(* PLC project Aufgabe2SPS, Beckhoff Automation GmbH TwinCAT PLC Control 3.5.13.20 *)
(* stored: creationDateTime 2020-03-31T15:44:23.6339566, modificationDateTime 2020-03-31T15:44:23.6389422 *)

TYPE ST_STATUS_WORD_DATA :
STRUCT
	inLenght : INT;
   overrunError  :  BOOL;
   framingError  :  BOOL;
   parityError  :  BOOL;
   bufferFull  :  BOOL;
   initAccepted  :  BOOL;
   receiveRequest  :  BOOL;
   transmitAccepted  :  BOOL;		

END_STRUCT
END_TYPE

TYPE ST_CurrentStatus :
STRUCT
	buttonYellow : BOOL;
	buttonBlue : BOOL;
	// usw...
END_STRUCT
END_TYPE

FUNCTION_BLOCK FB_EdgeDetector
VAR_INPUT
	b_InputSignal_k : BOOL;
END_VAR
VAR_OUTPUT
	b_PositiveEdge : BOOL;
	b_NegativeEdge : BOOL;
END_VAR
VAR
	b_InputSignal_k_1 : BOOL;
END_VAR

                  b_PositiveEdge := b_InputSignal_k AND NOT b_InputSignal_k_1;
b_NegativeEdge := NOT b_InputSignal_k AND b_InputSignal_k_1;

b_InputSignal_k_1 := b_InputSignal_k;
                
END_FUNCTION_BLOCK

FUNCTION F_AdditionFunction : INT
VAR_INPUT
	i_var1 : INT;
	i_var2 : INT;
END_VAR
VAR
	
END_VAR

                  F_AdditionFunction := i_var1 + i_var2;
                
END_FUNCTION

FUNCTION F_DivisionFunction : INT
VAR_INPUT
	i_var1 : INT;
	i_var2 : INT;
END_VAR
VAR
	
END_VAR

                  IF i_var2 = 0 THEN
	F_DivisionFunction := 0;
ELSE	
	F_DivisionFunction := i_var1 / i_var2;
END_IF

                
END_FUNCTION

FUNCTION F_STATUS_WORD_PROC : ST_STATUS_WORD_DATA
VAR_INPUT
	w_StatusWord : WORD;
END_VAR
VAR
END_VAR

                  

F_STATUS_WORD_PROC.transmitAccepted := w_StatusWord.0;
F_STATUS_WORD_PROC.parityError := w_StatusWord.1;
F_STATUS_WORD_PROC.initAccepted := w_StatusWord.2;
F_STATUS_WORD_PROC.bufferFull := w_StatusWord.3;
F_STATUS_WORD_PROC.parityError := w_StatusWord.4;
F_STATUS_WORD_PROC.framingError := w_StatusWord.5;
F_STATUS_WORD_PROC.overrunError := w_StatusWord.6;
F_STATUS_WORD_PROC.inLenght := WORD_TO_INT(SHR(w_StatusWord,8));
                
END_FUNCTION

PROGRAM MAIN
VAR
	// Lokale Variablen um die Funktionen
	// F_AdditionFunction und F_DivisionFunction zu testen
	i_var1   : INT;
	i_var2   : INT;
	i_addRes : INT;
	i_divRes : INT;
	
	// 16 bits
	w_myword : WORD := 16#5D7A;
	w_divRes : WORD;
	
	// 32 bits
	dw_mydword : DWORD;
	dw_mydword1 : DWORD;
	
	w_testWord : WORD;
	
	st_resRsProt : ST_STATUS_WORD_DATA;
	
	// Array von REAL, Dimension 10
	// arr_r_testArray : ARRAY[0..9] OF REAL;
	arr_r_testArray : ARRAY[1..10] OF REAL;
	
	// Variablen für FOR Schleife
	r_SummeArray : REAL;
	r_MulArray : REAL;
	
	// Variabel für FOR Schleife
	i_SchleifeIterVar : INT;
	
	// Edge detektor 2 Mal instanzieren
	fbEdgeDetectorGelb : FB_EdgeDetector;
	fbEdgeDetectorBlau : FB_EdgeDetector;
	
	// "Software" Taster um Edge Detektor zu testen
	bGelbTaster : BOOL;
	bBlauTaster : BOOL;
	
	// "Software" Leucthmelder
	bRedLight : BOOL;
	bGreenLight : BOOL;
	
	// Steuerbefehle für die Lampen
	bCommandForLights : BOOL := FALSE;
	
	// Number of Zyklen in 1/3 Sekunde (3 Hz)
	uiTicksNumber3Herz : UINT := 0;
	
	// Zähler
	uiTicksCounter : UINT := 0;
	
	// TRUE if positive Flanke bei gelbem Taster
	bGelbPositivEdge : BOOL;
	
	// Mittelwert vom Signal ***************
	rMeanVoltageValue : REAL;
	// Über die letzten 100 Werten
	rMeanVoltageValueForget : REAL;
	// Über die letzten 100 Werten mit Forgetting factor
	rMeanVoltageValueForgetWithRec : REAL;
	// Forgetting factor
	rLambda : REAL := 0.95;
	
	// Instanzieren Funktionsblock
	// Mittelwert mit rekursiven Anteil
	fbMeanWithRec : AverageCalculatorForgetBest;
	
	// Test-Variable mit Struktur
	stActStatus : ST_CurrentStatus;
END_VAR

                  // Aufruf Funktionen Addition/Division direkt vom Main
i_addRes := F_AdditionFunction(i_var1, i_var2);
i_divRes := F_DivisionFunction(i_var1, i_var2);

// Aufruf Funktionen Addition/Division direkt vom DoSomeMath
P_DoSomeMath.i_var1 := i_var1;
P_DoSomeMath.i_var2 := i_var2;
P_DoSomeMath();
i_addRes := P_DoSomeMath.i_addRes;
i_divRes := P_DoSomeMath.i_divRes;

// Teilung durch 8 -> shift right 3 bits
w_divRes := SHR(w_myword, 3);

// Multiplikation mit 8 -> shift left 3 bits
dw_mydword := SHL(w_myword, 3);

// Vier höchsten bits auf 1 setzen 
dw_mydword1 := dw_mydword OR 16#F0000000;

// Aufruf Funktion für RS232 Protokoll
// Auswertung vom Statuswort
st_resRsProt := F_STATUS_WORD_PROC(w_testWord);
 
// FOR Schleife um die Elemente von Array zusammen zu addieren
// bzw. zu multiplizieren
r_SummeArray := 0.0;
r_MulArray   := 1.0;
FOR i_SchleifeIterVar := 1 TO 10 DO
	r_SummeArray := r_SummeArray + arr_r_testArray[i_SchleifeIterVar];
	r_MulArray := r_MulArray * arr_r_testArray[i_SchleifeIterVar];
END_FOR


fbEdgeDetectorGelb(b_InputSignal_k := bGelbTaster);
bGelbPositivEdge := fbEdgeDetectorGelb.b_PositiveEdge;
// Alternativ, Funktionsausruf + Zuweisung Ergebnis in einem Schritt
// fbEdgeDetectorGelb(b_InputSignal_k := bGelbTaster, b_PositiveEdge => bGelbPositivEdge);
IF bGelbpositivEdge THEN
	// Hier Brekpoint setzen mit F9 um EdgeDetector zu testen
	r_MulArray := 0;
END_IF
 
fbEdgeDetectorBlau(b_InputSignal_k := bBlauTaster);

IF fbEdgeDetectorBlau.b_PositiveEdge THEN
	bCommandForLights := NOT bCommandForLights;
END_IF

IF bCommandForLights THEN
	uiTicksNumber3Herz := REAL_TO_UINT(1.0/3.0 / GVL_Constants.r_TaskTime);
	uiTicksCounter := uiTicksCounter + 1;
	IF uiTicksCounter = uiTicksNumber3Herz THEN
		uiTicksCounter := 0;	
		bRedLight := NOT bRedLight;
		bGreenLight := NOT bGreenLight;
	END_IF
END_IF

// Sensor simulieren !!
GVL_IO.intUltrasonicSensor := GVL_IO.intUltrasonicSensor + 100;
// -32768 -> 10 V, 32767 -> + 10 V
GVL_IO.voltageUltrasonicSensor := INT_TO_REAL(GVL_IO.intUltrasonicSensor) / 32767.0 * 10.0;

// Verschiebung nach links auf dem Buffer
ShifLeft();
// Letzte Spannung speichern
GVL_general.bufferArray[100] := GVL_IO.voltageUltrasonicSensor;

// Mittelwert
rMeanVoltageValue := AverageCalculator(GVL_general.bufferArray);
rMeanVoltageValueForget := AverageCalculatorForget(rLambda, GVL_general.bufferArray);

fbMeanWithRec(r_lambda := rLambda, 
	r_y_k := GVL_IO.voltageUltrasonicSensor,
	m_k => rMeanVoltageValueForgetWithRec); 
	


                
END_PROGRAM

PROGRAM P_DoSomeMath
VAR
END_VAR
// VAR_INPUT und VAR_OUTPUT müssen vor Hand
// hinzugefügt werden!!
VAR_INPUT
	i_var1 : INT;
	i_var2 : INT;
END_VAR
VAR_OUTPUT
	i_addRes : INT;
	i_divRes : INT;
END_VAR

                  
                
END_PROGRAM

FUNCTION ShifLeft : BOOL
VAR_INPUT
END_VAR
VAR
	iFor : INT;
END_VAR

                  FOR iFor := 1 TO 99 DO
	GVL_general.bufferArray[iFor] := GVL_general.bufferArray[iFor + 1];
END_FOR
                
END_FUNCTION

FUNCTION AverageCalculator : REAL
VAR_INPUT
	bufArr : ARRAY[1..100] OF REAL;
END_VAR
VAR
	iFor : INT;
END_VAR

                  AverageCalculator := 0.0;
FOR iFor := 1 TO 100 DO
	AverageCalculator := AverageCalculator + bufArr[iFor];
END_FOR
AverageCalculator  := AverageCalculator / 100;
                
END_FUNCTION

FUNCTION AverageCalculatorForget : REAL
VAR_INPUT
	rLambda : REAL := 0.95;
	bufArr : ARRAY[1..100] OF REAL;
END_VAR
VAR
	iFor : INT;
	rSumInter : REAL;
END_VAR

                  AverageCalculatorForget := 0.0;
rSumInter := 0.0;
FOR iFor := 1 TO 100 DO
	AverageCalculatorForget := AverageCalculatorForget + bufArr[iFor]*EXPT(rLambda,100-iFor);
	rSumInter := rSumInter + EXPT(rLambda,100-iFor);
END_FOR
AverageCalculatorForget  := AverageCalculatorForget / rSumInter;
                
END_FUNCTION

FUNCTION_BLOCK AverageCalculatorForgetBest
VAR_INPUT
	r_lambda : REAL;
	r_y_k : REAL;
END_VAR
VAR_OUTPUT
	m_k : REAL;
END_VAR
VAR
	m_k_1 : REAL;
END_VAR

                  m_k := r_lambda * m_k_1 + (1.0-r_lambda) * r_y_k;
m_k_1 := m_k;
                
END_FUNCTION_BLOCK

CONFIGURATION Application
  RESOURCE Aufgabe2SPS ON PLC
(* global variable list GVL_Constants *)
{attribute 'qualified_only'}
VAR_GLOBAL CONSTANT
	// Taskzeit 10 (ms)
	r_TaskTime : REAL := 0.01;
END_VAR
(* global variable list GVL_IO *)
{attribute 'qualified_only'}
VAR_GLOBAL
	intUltrasonicSensor AT %I* : INT;
	voltageUltrasonicSensor : REAL;
END_VAR
(* global variable list GVL_general *)
{attribute 'qualified_only'}
VAR_GLOBAL
	
	bufferArray : ARRAY[1..100] OF  REAL;
END_VAR
    TASK PlcTask(INTERVAL := T#0ms, PRIORITY := 20);
    PROGRAM MAIN WITH PlcTask : MAIN;
  END_RESOURCE
END_CONFIGURATION
